FUNCTION_BLOCK FB_AssemblyStation
VAR
    eState                  : E_AssemblyStationState := E_AssemblyStationState.Disabled;
    eFault                  : E_AssemblyStationFault := E_AssemblyStationFault.None;
    stStatusInternal        : ST_AssemblyStationStatus;
    stResult                : ST_ProcessResult;

    bStartRequest           : BOOL;
    bStopRequest            : BOOL;
    bResetRequest           : BOOL;

    tonMovementTimeout      : TON;
    tonActionDelay          : TON;
	tonGripperMismatch 		: TON;
    bSequenceActive         : BOOL;
END_VAR

METHOD PUBLIC Cyclic
VAR_INPUT
    bEnable                  : BOOL;
    bInitialising            : BOOL;

    bSafetyPermitted         : BOOL;
    bAirSupplySafe           : BOOL;
    bIndexReady              : BOOL;
    bIndexLocked             : BOOL;
    bIndexBusy               : BOOL;
    bAssemblySupportExtended : BOOL;

    bSlideExtended           : BOOL;
    bSlideRetracted          : BOOL;
    bGripperOpen             : BOOL;
    bGripperClosed           : BOOL;
    bRotationPick            : BOOL;
    bRotationPlace           : BOOL;

    tActionDelay             : TIME;
    tMovementTimeout         : TIME;
	tGripperMismatchDelay 	 : TIME := T#300MS;
	tReleaseDelay 			 : TIME;
	
END_VAR
VAR_OUTPUT
    bSlideExtendOutput       : BOOL;
    bSlideRetractOutput      : BOOL;
    bGripperOpenOutput       : BOOL;
    bGripperCloseOutput      : BOOL;
    bRotationPickOutput      : BOOL;
    bRotationPlaceOutput     : BOOL;
END_VAR
// =========================================================
// PHYSICAL ROTATION MAPPING
// =========================================================
// On this machine:
//   bRotationPick  / bRotationPickOutput  = physical 180 deg
//   bRotationPlace / bRotationPlaceOutput = physical 0 deg
//
// Required sequence:
// HOME 180 -> rotate 0 -> down -> close -> up ->
// rotate 180 -> down -> open -> up -> remain at 180.

// =========================================================
// OUTPUT DEFAULTS
// =========================================================
bSlideExtendOutput := FALSE;
bSlideRetractOutput := FALSE;
bGripperOpenOutput := FALSE;
bGripperCloseOutput := FALSE;
bRotationPickOutput := FALSE;
bRotationPlaceOutput := FALSE;

// =========================================================
// HOME STATUS
// =========================================================
stStatusInternal.bHome :=
    bSlideRetracted
    AND bGripperOpen
    AND bRotationPick;

// =========================================================
// SENSOR COHERENCE
// =========================================================
tonGripperMismatch(
    IN := bGripperOpen AND bGripperClosed,
    PT := tGripperMismatchDelay
);

IF bSlideExtended AND bSlideRetracted THEN
    eFault := E_AssemblyStationFault.SlideSensorMismatch;
    eState := E_AssemblyStationState.Fault;

ELSIF tonGripperMismatch.Q THEN
    eFault := E_AssemblyStationFault.GripperSensorMismatch;
    eState := E_AssemblyStationState.Fault;

ELSIF bRotationPick AND bRotationPlace THEN
    eFault := E_AssemblyStationFault.RotationSensorMismatch;
    eState := E_AssemblyStationState.Fault;
END_IF

// =========================================================
// RESET
// =========================================================
IF bResetRequest THEN
    bResetRequest := FALSE;
    bStartRequest := FALSE;
    bStopRequest := FALSE;
    tonMovementTimeout(IN := FALSE);
    tonActionDelay(IN := FALSE);

    IF NOT (bSlideExtended AND bSlideRetracted)
        AND NOT (bGripperOpen AND bGripperClosed)
        AND NOT (bRotationPick AND bRotationPlace)
    THEN
        eFault := E_AssemblyStationFault.None;
        eState := E_AssemblyStationState.Disabled;
        stResult.bValid := FALSE;
        stResult.bPassed := FALSE;
        stResult.eCode := E_ProcessResultCode.None;
        stResult.udiFaultCode := 0;
        stResult.sDetail := '';
    END_IF
END_IF

// =========================================================
// DISABLED / INITIALISING ENTRY
// =========================================================
IF eState <> E_AssemblyStationState.Fault THEN
    IF bInitialising THEN
        IF NOT bSlideRetracted THEN
            eState := E_AssemblyStationState.RecoveringSlideRetracted;
        ELSIF NOT bGripperOpen THEN
            eState := E_AssemblyStationState.RecoveringGripperOpen;
        ELSIF NOT bRotationPick THEN
            eState := E_AssemblyStationState.RecoveringRotationPlace;
        ELSE
            eState := E_AssemblyStationState.Idle;
        END_IF

    ELSIF bEnable AND eState = E_AssemblyStationState.Disabled THEN
        IF stStatusInternal.bHome THEN
            eState := E_AssemblyStationState.Idle;
        ELSE
            IF NOT bSlideRetracted THEN
                eState := E_AssemblyStationState.RecoveringSlideRetracted;
            ELSIF NOT bGripperOpen THEN
                eState := E_AssemblyStationState.RecoveringGripperOpen;
            ELSE
                eState := E_AssemblyStationState.RecoveringRotationPlace;
            END_IF
        END_IF

    ELSIF NOT bEnable THEN
        IF stStatusInternal.bHome THEN
            eState := E_AssemblyStationState.Disabled;
        END_IF
    END_IF
END_IF

// =========================================================
// STOP REQUEST
// =========================================================
IF bStopRequest AND eState <> E_AssemblyStationState.Fault THEN
    bStopRequest := FALSE;
    bStartRequest := FALSE;

    IF NOT bSlideRetracted THEN
        eState := E_AssemblyStationState.RecoveringSlideRetracted;
    ELSIF NOT bGripperOpen THEN
        eState := E_AssemblyStationState.RecoveringGripperOpen;
    ELSIF NOT bRotationPick THEN
        eState := E_AssemblyStationState.RecoveringRotationPlace;
    ELSE
        eState := E_AssemblyStationState.Idle;
    END_IF

    stResult.bValid := FALSE;
    stResult.bPassed := FALSE;
    stResult.eCode := E_ProcessResultCode.Aborted;
    stResult.sDetail := 'Assembly sequence stopped';
END_IF

// =========================================================
// ACTIVE-SEQUENCE PERMISSIVE SUPERVISION
// =========================================================
bSequenceActive :=
    (eState <> E_AssemblyStationState.Disabled)
    AND (eState <> E_AssemblyStationState.RecoveringSlideRetracted)
    AND (eState <> E_AssemblyStationState.RecoveringGripperOpen)
    AND (eState <> E_AssemblyStationState.RecoveringRotationPlace)
    AND (eState <> E_AssemblyStationState.Idle)
    AND (eState <> E_AssemblyStationState.Complete)
    AND (eState <> E_AssemblyStationState.Fault);

IF bSequenceActive THEN
    IF NOT bSafetyPermitted THEN
        eFault := E_AssemblyStationFault.SafetyLost;
        eState := E_AssemblyStationState.Fault;
    ELSIF NOT bAirSupplySafe THEN
        eFault := E_AssemblyStationFault.AirSupplyLost;
        eState := E_AssemblyStationState.Fault;
    ELSIF NOT bIndexReady OR NOT bIndexLocked OR bIndexBusy THEN
        eFault := E_AssemblyStationFault.IndexNotSafe;
        eState := E_AssemblyStationState.Fault;
    END_IF
END_IF

// =========================================================
// STATE MACHINE
// =========================================================
CASE eState OF

    E_AssemblyStationState.Disabled:
        tonMovementTimeout(IN := FALSE);
        tonActionDelay(IN := FALSE);

    // -----------------------------------------------------
    // RECOVERY TO HOME = 180 DEG
    // -----------------------------------------------------
    E_AssemblyStationState.RecoveringSlideRetracted:
        tonActionDelay(IN := FALSE);

        IF bAirSupplySafe AND bSafetyPermitted THEN
            bSlideRetractOutput := TRUE;
            tonMovementTimeout(IN := NOT bSlideRetracted, PT := tMovementTimeout);

            IF bSlideRetracted THEN
                tonMovementTimeout(IN := FALSE);

                IF NOT bGripperOpen THEN
                    eState := E_AssemblyStationState.RecoveringGripperOpen;
                ELSIF NOT bRotationPick THEN
                    eState := E_AssemblyStationState.RecoveringRotationPlace;
                ELSE
                    eState := E_AssemblyStationState.Idle;
                END_IF

            ELSIF tonMovementTimeout.Q THEN
                eFault := E_AssemblyStationFault.SlideRetractedSensorTimeout;
                eState := E_AssemblyStationState.Fault;
            END_IF
        ELSE
            tonMovementTimeout(IN := FALSE);
        END_IF

    E_AssemblyStationState.RecoveringGripperOpen:
        IF bAirSupplySafe AND bSafetyPermitted THEN
            tonMovementTimeout(IN := NOT bGripperOpen, PT := tMovementTimeout);
            bSlideRetractOutput := TRUE;
            bGripperOpenOutput := TRUE;

            IF bGripperOpen THEN
                tonMovementTimeout(IN := FALSE);

                IF NOT bRotationPick THEN
                    eState := E_AssemblyStationState.RecoveringRotationPlace;
                ELSE
                    eState := E_AssemblyStationState.Idle;
                END_IF

            ELSIF tonMovementTimeout.Q THEN
                eFault := E_AssemblyStationFault.GripperOpenSensorTimeout;
                eState := E_AssemblyStationState.Fault;
            END_IF
        ELSE
            tonMovementTimeout(IN := FALSE);
        END_IF

    E_AssemblyStationState.RecoveringRotationPlace:
        IF bAirSupplySafe AND bSafetyPermitted THEN
            tonMovementTimeout(IN := NOT bRotationPick, PT := tMovementTimeout);
            bSlideRetractOutput := TRUE;
            bGripperOpenOutput := TRUE;
            bRotationPickOutput := TRUE;

            IF bRotationPick THEN
                tonMovementTimeout(IN := FALSE);
                eState := E_AssemblyStationState.Idle;
            ELSIF tonMovementTimeout.Q THEN
                eFault := E_AssemblyStationFault.RotationPickSensorTimeout;
                eState := E_AssemblyStationState.Fault;
            END_IF
        ELSE
            tonMovementTimeout(IN := FALSE);
        END_IF

    // -----------------------------------------------------
    // READY / HOME = 180 DEG
    // -----------------------------------------------------
    E_AssemblyStationState.Idle:
        tonMovementTimeout(IN := FALSE);
        tonActionDelay(IN := FALSE);
        bSlideRetractOutput := TRUE;
        bGripperOpenOutput := TRUE;
        bRotationPickOutput := TRUE;

        IF bStartRequest THEN
            bStartRequest := FALSE;
            stResult.bValid := FALSE;
            stResult.bPassed := FALSE;
            stResult.eCode := E_ProcessResultCode.None;
            stResult.udiFaultCode := 0;
            stResult.sDetail := '';
			
			IF NOT bSafetyPermitted THEN
				eFault := E_AssemblyStationFault.SafetyLost;
				eState := E_AssemblyStationState.Fault;
			ELSIF NOT bAirSupplySafe THEN
				eFault := E_AssemblyStationFault.AirSupplyLost;
				eState := E_AssemblyStationState.Fault;
			ELSIF NOT bIndexReady OR NOT bIndexLocked OR bIndexBusy THEN
				eFault := E_AssemblyStationFault.IndexNotSafe;
				eState := E_AssemblyStationState.Fault;
			ELSIF NOT stStatusInternal.bHome THEN
				IF NOT bSlideRetracted THEN
					eState := E_AssemblyStationState.RecoveringSlideRetracted;
				ELSIF NOT bGripperOpen THEN
					eState := E_AssemblyStationState.RecoveringGripperOpen;
				ELSE
					eState := E_AssemblyStationState.RecoveringRotationPlace;
				END_IF
			ELSE
				eState := E_AssemblyStationState.RotatingToPick;
			END_IF
  
        END_IF

    // -----------------------------------------------------
    // 1. ROTATE FROM HOME 180 DEG TO PHYSICAL 0 DEG
    // -----------------------------------------------------
    E_AssemblyStationState.RotatingToPick:
        bSlideRetractOutput := TRUE;
        bGripperOpenOutput := TRUE;
        bRotationPlaceOutput := TRUE;
        tonMovementTimeout(IN := NOT bRotationPlace, PT := tMovementTimeout);

        IF bRotationPlace THEN
            tonMovementTimeout(IN := FALSE);
            eState := E_AssemblyStationState.DelayAfterRotateToPick;
        ELSIF tonMovementTimeout.Q THEN
            eFault := E_AssemblyStationFault.RotationPlaceSensorTimeout;
            eState := E_AssemblyStationState.Fault;
        END_IF

    E_AssemblyStationState.DelayAfterRotateToPick:
        bSlideRetractOutput := TRUE;
        bGripperOpenOutput := TRUE;
        bRotationPlaceOutput := TRUE;
        tonActionDelay(IN := TRUE, PT := tActionDelay);

        IF tonActionDelay.Q THEN
			tonActionDelay(IN := FALSE);
	
			IF bAssemblySupportExtended THEN
				eState := E_AssemblyStationState.ExtendingSlideToPick;
			END_IF
		END_IF

    // -----------------------------------------------------
    // 2. SLIDE DOWN AT PHYSICAL 0 DEG
    // -----------------------------------------------------
    E_AssemblyStationState.ExtendingSlideToPick:
        bSlideExtendOutput := TRUE;
        bGripperOpenOutput := TRUE;
        bRotationPlaceOutput := TRUE;
        tonMovementTimeout(IN := NOT bSlideExtended, PT := tMovementTimeout);

        IF bSlideExtended THEN
            tonMovementTimeout(IN := FALSE);
            eState := E_AssemblyStationState.DelayAfterPickExtend;
        ELSIF tonMovementTimeout.Q THEN
            eFault := E_AssemblyStationFault.SlideExtendedSensorTimeout;
            eState := E_AssemblyStationState.Fault;
        END_IF

    E_AssemblyStationState.DelayAfterPickExtend:
        bSlideExtendOutput := TRUE;
        bGripperOpenOutput := TRUE;
        bRotationPlaceOutput := TRUE;
        tonActionDelay(IN := TRUE, PT := tActionDelay);

        IF tonActionDelay.Q THEN
            tonActionDelay(IN := FALSE);
            eState := E_AssemblyStationState.ClosingGripper;
        END_IF

    // -----------------------------------------------------
    // 3. CLOSE GRIPPER AT PHYSICAL 0 DEG
    // -----------------------------------------------------
    E_AssemblyStationState.ClosingGripper:
        bSlideExtendOutput := TRUE;
        bGripperCloseOutput := TRUE;
        bRotationPlaceOutput := TRUE;
        tonMovementTimeout(IN := NOT bGripperClosed, PT := tMovementTimeout);

        IF bGripperClosed THEN
            tonMovementTimeout(IN := FALSE);
            eState := E_AssemblyStationState.DelayAfterGripperClose;
        ELSIF tonMovementTimeout.Q THEN
            eFault := E_AssemblyStationFault.GripperClosedSensorTimeout;
            eState := E_AssemblyStationState.Fault;
        END_IF

    E_AssemblyStationState.DelayAfterGripperClose:
        bSlideExtendOutput := TRUE;
        bGripperCloseOutput := TRUE;
        bRotationPlaceOutput := TRUE;
        tonActionDelay(IN := TRUE, PT := tActionDelay);

        IF tonActionDelay.Q THEN
            tonActionDelay(IN := FALSE);
            eState := E_AssemblyStationState.RetractingSlideWithPart;
        END_IF

    // -----------------------------------------------------
    // 4. SLIDE UP WITH PART AT PHYSICAL 0 DEG
    // -----------------------------------------------------
    E_AssemblyStationState.RetractingSlideWithPart:
        bSlideRetractOutput := TRUE;
        bGripperCloseOutput := TRUE;
        bRotationPlaceOutput := TRUE;
        tonMovementTimeout(IN := NOT bSlideRetracted, PT := tMovementTimeout);

        IF bSlideRetracted THEN
            tonMovementTimeout(IN := FALSE);
            eState := E_AssemblyStationState.DelayAfterPickRetract;
        ELSIF tonMovementTimeout.Q THEN
            eFault := E_AssemblyStationFault.SlideRetractedSensorTimeout;
            eState := E_AssemblyStationState.Fault;
        END_IF

    E_AssemblyStationState.DelayAfterPickRetract:
        bSlideRetractOutput := TRUE;
        bGripperCloseOutput := TRUE;
        bRotationPlaceOutput := TRUE;
        tonActionDelay(IN := TRUE, PT := tActionDelay);

        IF tonActionDelay.Q THEN
            tonActionDelay(IN := FALSE);
            eState := E_AssemblyStationState.RotatingToPlace;
        END_IF

    // -----------------------------------------------------
    // 5. ROTATE WITH PART TO PHYSICAL 180 DEG
    // -----------------------------------------------------
    E_AssemblyStationState.RotatingToPlace:
        bSlideRetractOutput := TRUE;
        bGripperCloseOutput := TRUE;
        bRotationPickOutput := TRUE;
        tonMovementTimeout(IN := NOT bRotationPick, PT := tMovementTimeout);

        IF bRotationPick THEN
            tonMovementTimeout(IN := FALSE);
            eState := E_AssemblyStationState.DelayAfterRotateToPlace;
        ELSIF tonMovementTimeout.Q THEN
            eFault := E_AssemblyStationFault.RotationPickSensorTimeout;
            eState := E_AssemblyStationState.Fault;
        END_IF

    E_AssemblyStationState.DelayAfterRotateToPlace:
        bSlideRetractOutput := TRUE;
        bGripperCloseOutput := TRUE;
        bRotationPickOutput := TRUE;
        tonActionDelay(IN := TRUE, PT := tActionDelay);

        IF tonActionDelay.Q THEN
            tonActionDelay(IN := FALSE);
            eState := E_AssemblyStationState.ExtendingSlideToPlace;
        END_IF

    // -----------------------------------------------------
    // 6. SLIDE DOWN AT PHYSICAL 180 DEG
    // -----------------------------------------------------
    E_AssemblyStationState.ExtendingSlideToPlace:
        bSlideExtendOutput := TRUE;
        bGripperCloseOutput := TRUE;
        bRotationPickOutput := TRUE;
        tonMovementTimeout(IN := NOT bSlideExtended, PT := tMovementTimeout);

        IF bSlideExtended THEN
            tonMovementTimeout(IN := FALSE);
            eState := E_AssemblyStationState.DelayAfterPlaceExtend;
        ELSIF tonMovementTimeout.Q THEN
            eFault := E_AssemblyStationFault.SlideExtendedSensorTimeout;
            eState := E_AssemblyStationState.Fault;
        END_IF

    E_AssemblyStationState.DelayAfterPlaceExtend:
        bSlideExtendOutput := TRUE;
        bGripperCloseOutput := TRUE;
        bRotationPickOutput := TRUE;
        tonActionDelay(IN := TRUE, PT := tReleaseDelay);

        IF tonActionDelay.Q THEN
            tonActionDelay(IN := FALSE);
            eState := E_AssemblyStationState.OpeningGripper;
        END_IF

    // -----------------------------------------------------
    // 7. OPEN GRIPPER AT PHYSICAL 180 DEG
    // -----------------------------------------------------
    E_AssemblyStationState.OpeningGripper:
        bSlideExtendOutput := TRUE;
        bGripperOpenOutput := TRUE;
        bRotationPickOutput := TRUE;
        tonMovementTimeout(IN := NOT bGripperOpen, PT := tMovementTimeout);

        IF bGripperOpen THEN
            tonMovementTimeout(IN := FALSE);
            eState := E_AssemblyStationState.DelayAfterGripperOpen;
        ELSIF tonMovementTimeout.Q THEN
            eFault := E_AssemblyStationFault.GripperOpenSensorTimeout;
            eState := E_AssemblyStationState.Fault;
        END_IF

    E_AssemblyStationState.DelayAfterGripperOpen:
        bSlideExtendOutput := TRUE;
        bGripperOpenOutput := TRUE;
        bRotationPickOutput := TRUE;
        tonActionDelay(IN := TRUE, PT := tActionDelay);

        IF tonActionDelay.Q THEN
            tonActionDelay(IN := FALSE);
            eState := E_AssemblyStationState.RetractingSlideHome;
        END_IF

    // -----------------------------------------------------
    // 8. SLIDE UP AND REMAIN AT PHYSICAL 180 DEG
    // -----------------------------------------------------
    E_AssemblyStationState.RetractingSlideHome:
        bSlideRetractOutput := TRUE;
        bGripperOpenOutput := TRUE;
        bRotationPickOutput := TRUE;
        tonMovementTimeout(IN := NOT bSlideRetracted, PT := tMovementTimeout);

        IF bSlideRetracted THEN
            tonMovementTimeout(IN := FALSE);
            eState := E_AssemblyStationState.DelayAfterHomeRetract;
        ELSIF tonMovementTimeout.Q THEN
            eFault := E_AssemblyStationFault.SlideRetractedSensorTimeout;
            eState := E_AssemblyStationState.Fault;
        END_IF

    E_AssemblyStationState.DelayAfterHomeRetract:
        bSlideRetractOutput := TRUE;
        bGripperOpenOutput := TRUE;
        bRotationPickOutput := TRUE;
        tonActionDelay(IN := TRUE, PT := tActionDelay);

        IF tonActionDelay.Q THEN
            tonActionDelay(IN := FALSE);
            stResult.bValid := TRUE;
            stResult.bPassed := TRUE;
            stResult.eCode := E_ProcessResultCode.Pass;
            stResult.udiFaultCode := 0;
            stResult.sDetail := 'Barrel flipping and assembly sequence complete';
            eState := E_AssemblyStationState.Complete;
        END_IF

    E_AssemblyStationState.Complete:
        bSlideRetractOutput := TRUE;
        bGripperOpenOutput := TRUE;
        bRotationPickOutput := TRUE;
        tonMovementTimeout(IN := FALSE);
        tonActionDelay(IN := FALSE);

    E_AssemblyStationState.Fault:
        tonMovementTimeout(IN := FALSE);
        tonActionDelay(IN := FALSE);
		stResult.bValid := FALSE;
    	stResult.bPassed := FALSE;

END_CASE

// =========================================================
// PUBLIC STATUS
// =========================================================
stStatusInternal.eState := eState;
stStatusInternal.eFault := eFault;
stStatusInternal.bReady := eState = E_AssemblyStationState.Idle;
stStatusInternal.bDone := eState = E_AssemblyStationState.Complete;
stStatusInternal.bFaulted := eState = E_AssemblyStationState.Fault;

stStatusInternal.bBusy :=
    bSequenceActive
    OR (eState = E_AssemblyStationState.RecoveringSlideRetracted)
    OR (eState = E_AssemblyStationState.RecoveringGripperOpen)
    OR (eState = E_AssemblyStationState.RecoveringRotationPlace);

stStatusInternal.bIndexPermissive :=
    stStatusInternal.bHome
    AND NOT stStatusInternal.bBusy
    AND NOT stStatusInternal.bFaulted;

stStatusInternal.bSlideRetracted := bSlideRetracted;
stStatusInternal.bSlideExtended := bSlideExtended;
stStatusInternal.bGripperOpen := bGripperOpen;
stStatusInternal.bGripperClosed := bGripperClosed;
stStatusInternal.bRotationPick := bRotationPick;
stStatusInternal.bRotationPlace := bRotationPlace;

// =========================================================
// STATUS MESSAGE
// =========================================================
CASE eState OF
    E_AssemblyStationState.Disabled:
        stStatusInternal.sMessage := 'Assembly station disabled';

    E_AssemblyStationState.RecoveringSlideRetracted:
        stStatusInternal.sMessage := 'Assembly station homing - retracting transfer slide';

    E_AssemblyStationState.RecoveringGripperOpen:
        stStatusInternal.sMessage := 'Assembly station homing - opening rotary gripper';

    E_AssemblyStationState.RecoveringRotationPlace:
        stStatusInternal.sMessage := 'Assembly station homing - rotating gripper to 180 degrees';

    E_AssemblyStationState.Idle:
        stStatusInternal.sMessage := 'Assembly station ready at 180 degree home position';

    E_AssemblyStationState.RotatingToPick:
        stStatusInternal.sMessage := 'Assembly station - rotating gripper from 180 to 0 degree pick position';

    E_AssemblyStationState.DelayAfterRotateToPick:
        stStatusInternal.sMessage := 'Assembly station - 0 degree pick position settling';

    E_AssemblyStationState.ExtendingSlideToPick:
        stStatusInternal.sMessage := 'Assembly station - lowering slide to pick barrel';

    E_AssemblyStationState.DelayAfterPickExtend:
        stStatusInternal.sMessage := 'Assembly station - pick position settling';

    E_AssemblyStationState.ClosingGripper:
        stStatusInternal.sMessage := 'Assembly station - closing gripper';

    E_AssemblyStationState.DelayAfterGripperClose:
        stStatusInternal.sMessage := 'Assembly station - gripper settling';

    E_AssemblyStationState.RetractingSlideWithPart:
        stStatusInternal.sMessage := 'Assembly station - lifting barrel';

    E_AssemblyStationState.DelayAfterPickRetract:
        stStatusInternal.sMessage := 'Assembly station - lift position settling';

    E_AssemblyStationState.RotatingToPlace:
        stStatusInternal.sMessage := 'Assembly station - rotating barrel to 180 degrees';

    E_AssemblyStationState.DelayAfterRotateToPlace:
        stStatusInternal.sMessage := 'Assembly station - 180 degree position settling';

    E_AssemblyStationState.ExtendingSlideToPlace:
        stStatusInternal.sMessage := 'Assembly station - lowering barrel to assembly position';

    E_AssemblyStationState.DelayAfterPlaceExtend:
        stStatusInternal.sMessage := 'Assembly station - assembly position settling';

    E_AssemblyStationState.OpeningGripper:
        stStatusInternal.sMessage := 'Assembly station - releasing barrel';

    E_AssemblyStationState.DelayAfterGripperOpen:
        stStatusInternal.sMessage := 'Assembly station - release settling';

    E_AssemblyStationState.RetractingSlideHome:
        stStatusInternal.sMessage := 'Assembly station - retracting transfer slide';

    E_AssemblyStationState.DelayAfterHomeRetract:
        stStatusInternal.sMessage := 'Assembly station - home height settling';

    E_AssemblyStationState.Complete:
        stStatusInternal.sMessage := 'Assembly station cycle complete';

    E_AssemblyStationState.Fault:
        stStatusInternal.sMessage := 'Assembly station fault';
END_CASE
END_METHOD

METHOD PUBLIC GetResult : ST_ProcessResult
VAR_INPUT
END_VAR
GetResult := stResult;
END_METHOD

METHOD PUBLIC GetStatus : ST_AssemblyStationStatus
VAR_INPUT
END_VAR
GetStatus := stStatusInternal;
END_METHOD

METHOD PUBLIC IndexPermissive : BOOL
VAR_INPUT
END_VAR
IndexPermissive := stStatusInternal.bIndexPermissive;
END_METHOD

METHOD PUBLIC IsBusy : BOOL
VAR_INPUT
END_VAR
IsBusy := stStatusInternal.bBusy;
END_METHOD

METHOD PUBLIC IsDone : BOOL
VAR_INPUT
END_VAR
IsDone := stStatusInternal.bDone;
END_METHOD

METHOD PUBLIC IsFaulted : BOOL
VAR_INPUT
END_VAR
IsFaulted := stStatusInternal.bFaulted;
END_METHOD

METHOD PUBLIC IsHome : BOOL
VAR_INPUT
END_VAR
IsHome := stStatusInternal.bHome;
END_METHOD

METHOD PUBLIC IsReady : BOOL
VAR_INPUT
END_VAR
IsReady := stStatusInternal.bReady;
END_METHOD

METHOD PUBLIC RequestReset
VAR_INPUT
END_VAR
bResetRequest := TRUE;
END_METHOD

METHOD PUBLIC RequestStart : BOOL
VAR_INPUT
END_VAR
RequestStart := FALSE;
IF eState = E_AssemblyStationState.Idle
    AND NOT stStatusInternal.bFaulted
THEN
    bStartRequest := TRUE;
    RequestStart := TRUE;
END_IF
END_METHOD

METHOD PUBLIC RequestStop
VAR_INPUT
END_VAR
bStopRequest := TRUE;
END_METHOD

METHOD PUBLIC Reset
VAR_INPUT
END_VAR
bResetRequest := TRUE;
END_METHOD

END_FUNCTION_BLOCK

(* stored: Version 1.1.0.1, ProductVersion 3.1.4026.18
   POU FB_AssemblyStation: Id {eebba9b2-d3c3-4ba3-a9e5-6f547c7e9dc1}, SpecialFunc None
   Method Cyclic: Id {51267cf8-e399-4cca-8ccc-e5e546c24a74}
   Method GetResult: Id {65738071-41c4-48f0-abc5-664e3fc87d0e}
   Method GetStatus: Id {e00fe120-fbbd-49b5-8d7b-6d2aaadb62c6}
   Method IndexPermissive: Id {06e09253-7ec3-473e-aec8-62b55e58cb22}
   Method IsBusy: Id {ff9f5262-4c3c-4172-9c67-4c7d0cda04de}
   Method IsDone: Id {b622034e-cb59-4a37-85ed-758047f9fdd6}
   Method IsFaulted: Id {135bd38f-c2f5-49af-b71f-33f31fa75006}
   Method IsHome: Id {78926916-e1af-476d-abc4-a0cf4aa15cfa}
   Method IsReady: Id {d494cff0-1b76-4be8-a234-462b06ac6efc}
   Method RequestReset: Id {ca408c3f-ace4-42a7-93a1-ea3f25d9d23f}
   Method RequestStart: Id {b709cea2-7aee-43ce-b498-1c542bf332e4}
   Method RequestStop: Id {df0ec237-cccc-444f-a3e7-ac95231686e0}
   Method Reset: Id {0a767d47-1b65-4608-9e88-4d1f6f2cb7ce} *)
